PROGRAM pouMsgS6
VAR
	
	
	
END_VAR

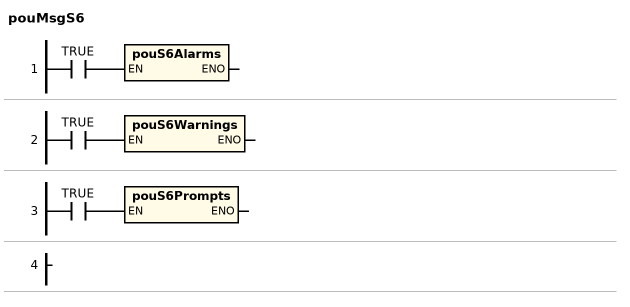
// NETWORK 1
pouS6Alarms();

// NETWORK 2
pouS6Warnings();

// NETWORK 3
pouS6Prompts();

// NETWORK 4

END_PROGRAM

(* stored: Version 1.1.0.1, ProductVersion 3.1.4024.12
   POU pouMsgS6: Id {e37d8473-1ec8-43ea-80a0-228dd5d4479d}, SpecialFunc None *)
